ABB RAPID module: Wobj_base_mm_concrete1.mod

MODULE Wobj_base_mm_concrete1
	! Points are read in order of declaration.
  ! Please do not change the order of points!

  LOCAL PERS robtarget pWobj_U_PointX1:=[[1087.932,613.0908,-509.424],[0.00214569480158389,-0.517328083515167,-0.855783462524414,0.00129179819487035],[0,0,1,0],[9E+09,9E+09,9E+09,9E+09,9E+09,9E+09]];
	LOCAL PERS robtarget pWobj_U_PointX2:=[[1100.739,-569.2292,-509.4458],[0.00218031578697264,-0.517317712306976,-0.855789661407471,0.00129661557730287],[-1,-1,0,0],[9E+09,9E+09,9E+09,9E+09,9E+09,9E+09]];
	LOCAL PERS robtarget pWobj_U_PointY1:=[[1845.216,622.8621,-508.772],[0.00218978128395975,-0.517311751842499,-0.855793178081512,0.00131216901354492],[0,0,0,0],[9E+09,9E+09,9E+09,9E+09,9E+09,9E+09]];

ENDMODULE
